FUNCTION_BLOCK FB_DCSystem EXTENDS FB_SystemContinous
VAR_INPUT
END_VAR
VAR_OUTPUT
END_VAR
VAR
	//default parameters
	localDefaultParameters : ST_DCSystemDefaultParameters;
	
	//pumps
	stPU245DefaultParameters : ST_PumpGrundfosMagna3DefaultParameters := (bPumpBeforeApplication := FALSE, tTaskCycleTime := GlobalVariables.tTaskCycleTime_MAIN, tCtrlCycleTime := GlobalVariables.tCtrlCycleTime_MAIN);
	PU245 : FB_PumpGrundfosMagna3 := (ST_DefaultParameters := stPU245DefaultParameters);;

	//valves
	stSV245DefaultParameters : ST_DiscreteValveDefaultParameters := (nFeedback := 0);
	SV245 : FB_DiscreteValve := (ST_DefaultParameters := stSV245DefaultParameters);
	
	WMZ245 : FB_MollineEHeatCounter;
	
	//internal variables
	bSetStatusOn_PU245 : BOOL;
	bSetStatusOn_SV245 : BOOL;
	
	//timer
	bStartTimer : BOOL;
	Timer : TON;
END_VAR

MAIN();

//use timer because valve has no feedback signal (75 sec)
Timer(IN := bStartTimer,
	PT := T#75S);

SV245.GetState_BI();
SV245(bSetStatusOnAutomatic := bSetStatusOn_SV245,
	bAlgorithmPermission := bAlgorithmPermission);
SV245.SetState_BO();

//pump controls return temperature
PU245.GetState_Profibus();
PU245(bSetStatusOnAutomatic := bSetStatusOn_PU245,
	bAlgorithmPermission := bAlgorithmPermission,
	fSetPointAutomatic := fSetPoint,
	fThermalPowerExternal := WMZ245.fHeatFlowRate,
	nControlModeAutomatic := 3);
PU245.SetState_Profibus();

WMZ245(aHeatCounterTelegramm := aTelegramm_WMZ245);

METHOD PROTECTED  CheckError : BOOL
VAR_INPUT
END_VAR
VAR_OUTPUT
	bError : BOOL;
END_VAR
IF PU245.bError THEN
	bError := TRUE;
END_IF
END_METHOD

METHOD PROTECTED  Operational : BOOL
VAR_INPUT
END_VAR
VAR_OUTPUT
	bSwitchToWorking : BOOL := FALSE;
END_VAR
bSetStatusOn_PU245 := TRUE;

IF PU245.bStatusOn THEN
	bSwitchToWorking := TRUE;
END_IF
END_METHOD

METHOD PROTECTED  RampDown : BOOL
VAR_INPUT
END_VAR
VAR_OUTPUT
	bRampDownFinished : BOOL := FALSE;
END_VAR
bSetStatusOn_PU245 := FALSE;

IF NOT PU245.bStatusOn THEN
	bSetStatusOn_SV245 := FALSE;
	bStartTimer := TRUE;
	IF Timer.Q THEN
		bStartTimer := FALSE;
		bRampDownFinished := TRUE;
	END_IF
END_IF
END_METHOD

METHOD PROTECTED  RampUp : BOOL
VAR_INPUT
END_VAR
VAR_OUTPUT
	bRampUpFinished : BOOL := FALSE;
END_VAR
bSetStatusOn_SV245 := TRUE;
bStartTimer := TRUE;

IF Timer.Q THEN
	bStartTimer := FALSE;
	bRampUpFinished := TRUE;
END_IF
END_METHOD

METHOD PROTECTED   SetSetPointLimits : BOOL
VAR_INPUT
END_VAR
IF  PU245.nControlModeAutomatic = 3 THEN
	aSetPointLimits[1] := localDefaultParameters.aSetPointLimitsTemperatureDifference[1];
	aSetPointLimits[2] := localDefaultParameters.aSetPointLimitsTemperatureDifference[2];
ELSE
	aSetPointLimits[1] := localDefaultParameters.aSetPointLimitsRelativeSpeed[1];
	aSetPointLimits[2] := localDefaultParameters.aSetPointLimitsRelativeSpeed[2];
END_IF
END_METHOD

METHOD PROTECTED  SetState : BOOL
VAR_INPUT
END_VAR
VAR_OUTPUT
END_VAR
fOperatingPoint := PU245.localState.fTemperatureDifference;

controlState.bStatusOn := bSetStatusOn;
setPointState.aSetPointLimits := aSetPointLimits;
setPointState.fSetPoint := fSetPoint;
setPointState.fOperatingPoint := fOperatingPoint;
setPointState.sSetPointUnit := 'K';
setPointState.sOperatingPointUnit := 'K';
END_METHOD

METHOD PROTECTED  Working : BOOL
VAR_INPUT
END_VAR
VAR_OUTPUT
	bSwitchToOperational : BOOL := FALSE;
END_VAR
//empty method
END_METHOD

END_FUNCTION_BLOCK

(* stored: Version 1.1.0.1, ProductVersion 3.1.4024.10
   POU FB_DCSystem: Id {9dbe8672-d93a-4703-8594-a33cc1d0c6c6}, SpecialFunc None
   Method CheckError: Id {335c28ac-45c3-487e-8d10-7aaec001f52a}
   Method Operational: Id {804b0cb9-bb45-40d5-8185-14247aa58afb}
   Method RampDown: Id {02e065ee-2516-444f-bbf9-1fa5c4e69c5c}
   Method RampUp: Id {d124129b-1537-4d55-bd40-13f9ebefeb89}
   Method SetSetPointLimits: Id {ace4869b-5552-4ded-8639-24c5baab0e11}
   Method SetState: Id {649d5ace-5c25-4698-a64e-e4990d28bd12}
   Method Working: Id {f5cd3651-4a32-4fda-a3f3-7690d2939edf} *)
